(* Logix 5000 project; controller WWTP_SEC_CLX vendor 1 type 14 code 54 rev 17.2; software revision 17.00; part 9 of 13 *)
(* tags used below, declared in another part *)
   Inp_Faulted : BOOL;   // 1=Drive has Faulted (see drive display or manual)
   Inp_IntlkOK : BOOL;   // 1=Interlocks OK, drive can start/run
   Inp_NBIntlkOK : BOOL;   // 1=Non-Bypassable Interlocks OK, drive can start/run
   Inp_IOFault : BOOL;   // Input Communication Status 0=OK, 1=fail
   Inp_Sim : BOOL;   // 1=Simulate working drive; 0=Start/Stop/ Monitor actual drive
   Inp_Reset : BOOL;   // 1=Reset drive fault conditions and latched Alarms
   Cfg_HasOutDatalink : BOOL;   // 1=A signal is connected to Out_Datalink1
   Cfg_PCmdClear : BOOL;   // 1=Clear Program Commands on receipt 0=Leave Set
   Cfg_OvrdPermIntlk : BOOL;   // 1=Override ignores Bypassable Perm/ Intlk; 0=always use Perm/Intlk
   Cfg_HasFailToStartAlm : BOOL;   // 1=Fail to Start Alarm exists and will be checked
   Cfg_HasFailToStopAlm : BOOL;   // 1=Fail to Stop Alarm exists and will be checked
   Cfg_HasIntlkTripAlm : BOOL;   // 1=Interlock Trip Alarm exists and will be checked
   Cfg_HasDriveFaultAlm : BOOL;   // 1=Drive Fault alarm exists and will be checked
   Cfg_HasIOFaultAlm : BOOL;   // 1=I/O Fault Alarm exists and will be checked
   Cfg_FailToStartResetReqd : BOOL;   // 1=Reset requied to clear Fail to Start Alarm
   Cfg_FailToStopResetReqd : BOOL;   // 1=Reset required to clear Fail to Stop Alarm
   Cfg_IntlkTripResetReqd : BOOL;   // 1=Reset required to clear Interlock Trip Alarm
   Cfg_DriveFaultResetReqd : BOOL;   // 1=Reset required to clear Drive Fault Alarm
   Cfg_IOFaultResetReqd : BOOL;   // 1=Reset required to clear I/O Fault Alarm
   Cfg_FailToStartAckReqd : BOOL;   // 1=Acknowledge required for Fail to Start Alarm
   Cfg_FailToStopAckReqd : BOOL;   // 1=Acknowledge required for Fail to Stop Alarm
   Cfg_IntlkTripAckReqd : BOOL;   // 1=Acknowledge required for Interlock Trip Alarm
   Cfg_DriveFaultAckReqd : BOOL;   // 1=Acknowledge required for Drive Fault Alarm
   Cfg_IOFaultAckReqd : BOOL;   // 1=Acknowledge required for I/O Fault Alarm
   Cfg_FailToStartSeverity : SINT;   // Fail To Start Alarm Severity 1=info 2=warn 3=excep 4=fault
   Cfg_FailToStopSeverity : SINT;   // Fail To Stop Alarm Severity 1=info 2=warn 3=excep 4=fault
   Cfg_IntlkTripSeverity : SINT;   // Interlock Trip Alarm Severity 1=info 2=warn 3=excep 4=fault
   Cfg_DriveFaultSeverity : SINT;   // Drive Fault Alarm Severity 1=info, 2=warn, 3=excep, 4=fault
   Cfg_IOFaultSeverity : SINT;   // I/O Fault Alarm Severity 1=info 2=warn 3=excep 4=fault
   Cfg_MinSpdRef : REAL;   // Minimum Speed Reference in EU (for limiting)
   Cfg_MaxSpdRef : REAL;   // Maximum Speed Reference in EU (for limiting)
   Cfg_SpeedRefRawMin : INT;   // Speed Reference Minimum in Drive (raw) Units (for scaling)
   Cfg_SpeedRefRawMax : INT;   // Speed Reference Maximum in Drive (raw) Units (for scaling)
   Cfg_SpeedRefEUMin : REAL;   // Speed Reference Minimum in Engineering Units (for scaling)
   Cfg_SpeedRefEUMax : REAL;   // Speed Reference Maximum in Engineering Units (for scaling)
   Cfg_SpeedFdbkRawMin : INT;   // Speed Feedback Minimum in Drive (raw) Units (for scaling)
   Cfg_SpeedFdbkRawMax : INT;   // Speed Feedback Maximum in Drive (raw) Units (for scaling)
   Cfg_SpeedFdbkEUMin : REAL;   // Speed Feedback Minimum in Engineering Units (for scaling)
   Cfg_SpeedFdbkEUMax : REAL;   // Speed Feedback Maximum in Engineering Units (for scaling)
   Cfg_InpDatalinkRawMin : INT;   // Input Datalink Minimum in Drive (raw) Units (for scaling)
   Cfg_InpDatalinkRawMax : INT;   // Input Datalink Maximum in Drive (raw) Units (for scaling)
   Cfg_InpDatalinkEUMin : REAL;   // Input Datalink Minimum in Engineering Units (for scaling)
   Cfg_InpDatalinkEUMax : REAL;   // Input Datalink Maximum in Engineering Units (for scaling)
   Cfg_OutDatalinkMin : REAL;   // Minimum Output Datalink in EU (for limiting)
   Cfg_OutDatalinkMax : REAL;   // Maximum Output Datalink in EU (for limiting)
   Cfg_OutDatalinkRawMin : INT;   // Output Datalink Minimum in Drive (raw) Units (for scaling)
   Cfg_OutDatalinkRawMax : INT;   // Output Datalink Maximum in Drive (raw) Units (for scaling)
   Cfg_OutDatalinkEUMin : REAL;   // Output Datalink Minimum in Engineering Units (for scaling)
   Cfg_OutDatalinkEUMax : REAL;   // Output Datalink Maximum in Engineering Units (for scaling)
   PCmd_Reset : BOOL;   // Program Command to Reset drive fault and all Alarms requiring Reset
   PCmd_FailToStartAck : BOOL;   // Program Command to Acknowledge Fail to Start Alarm
   PCmd_FailToStartInhibit : BOOL;   // Program Command to Inhibit Fail to Start Alarm
   PCmd_FailToStartUninhibit : BOOL;   // Program Command to Uninhibit Fail to Start Alarm
   PCmd_FailToStopAck : BOOL;   // Program Command to Acknowledge Fail to Stop Alarm
   PCmd_FailToStopInhibit : BOOL;   // Program Command to Inhibit Fail to Stop Alarm
   PCmd_FailToStopUninhibit : BOOL;   // Program Command to Uninhibit Fail to Stop Alarm
   PCmd_IntlkTripAck : BOOL;   // Program Command to Acknowledge Interlock Trip Alarm
   PCmd_IntlkTripInhibit : BOOL;   // Program Command to Inhibit Interlock Trip Alarm
   PCmd_IntlkTripUninhibit : BOOL;   // Program Command to Uninhibit Interlock Trip Alarm
   PCmd_DriveFaultAck : BOOL;   // Program Command to Acknowledge Drive Fault Alarm
   PCmd_DriveFaultInhibit : BOOL;   // Program Command to Inhibit Drive Fault Alarm
   PCmd_DriveFaultUninhibit : BOOL;   // Program Command to Uninhibit Drive Fault Alarm
   PCmd_IOFaultAck : BOOL;   // Program Command to Acknowledge I/O Fault Alarm
   PCmd_IOFaultInhibit : BOOL;   // Program Command to Inhibit I/O Fault Alarm
   PCmd_IOFaultUninhibit : BOOL;   // Program Command to Uninhibit I/O Fault Alarm
   OCmd_Reset : BOOL;   // Operator Command to Reset all Alarms requiring Reset
   Out_SpeedRef : INT;   // Drive Speed Reference in Drive Units (typ. 0-32767 = 0 to max freq.)
   Out_Datalink : INT;   // Auxiliary Signal (datalink) Output in Drive (raw) Units
   Out_Run : BOOL;   // 1=Start/Run Drive, 0=Stop Drive (for held starter type)
   Out_Stop : BOOL;   // 1=Stop Drive, 0=drive left in current state
   Out_Start : BOOL;   // 1=Start Drive, 0=drive left in current state
   Out_Jog : BOOL;   // 1=Jog drive at Jog Speed, -->0=stop jogging
   Out_ClearFault : BOOL;   // 1=Attempt to clear Drive Fault
   Out_Fwd : BOOL;   // 1=Set drive direction to Forward
   Out_Rev : BOOL;   // 1=Set drive direction to Reverse
   Val_Notify : SINT;   // Current Alarm Level and Acknowledgement (enumeration)
   Sts_Disabled : BOOL;   // 1=Drive is Disabled
   Sts_Err : BOOL;   // 1=Error in Config: see detail bits for reason
   Err_Timer : BOOL;   // 1=Error in Config: Invalid Check or Reset Pulse Time (use 0 to 2147483)
   Err_Sim : BOOL;   // 1=Error in Config: simulation timer preset: use 0 to 2147483)
   Err_Alarm : BOOL;   // 1=Error in Config: Invalid Alarm Severity
   Err_FdbkRaw : BOOL;   // 1=Erron in Config: Speed Fdbk Raw Min = Max
   Err_FdbkEU : BOOL;   // 1=Error in Config: Speed Fdbk EU Min = Max
   Err_RefLim : BOOL;   // 1=Error in Config: Speed Ref Limit Min > Max
   Err_RefEU : BOOL;   // 1=Error in Config: Speed Ref EU Min = Max
   Err_RefRaw : BOOL;   // 1=Error in Config: Speed Ref Raw Min = Max
   Err_InpDLRaw : BOOL;   // 1=Error in Config: Input Datalink Raw Min = Max
   Err_InpDLEU : BOOL;   // 1=Error in Config: Input Datalink EU Min = Max
   Err_OutDLLim : BOOL;   // 1=Error in Config: Output Datalink Limits Min > Max
   Err_OutDLEU : BOOL;   // 1=Error in Config: Output Datalink EU Min = Max
   Err_OutDLRaw : BOOL;   // 1=Error in Config: Output Datalink Raw Min = Max
   Sts_Hand : BOOL;   // 1=Mode is Hand (supersedes Maint, Ovrd, Prog, Oper)
   Sts_Maint : BOOL;   // 1=Mode is Maintenance (supersedes Ovrd, Prog, Oper)
   Sts_Ovrd : BOOL;   // 1=Mode is Override (supersedes Prog, Oper)
   Sts_Prog : BOOL;   // 1=Mode is Program (auto)
   Sts_Oper : BOOL;   // 1=Mode is Operator (manual)
   Sts_ProgOperLock : BOOL;   // 1=Program or Operator has requested Mode Lock
   Sts_FailToStart : BOOL;   // 1=Drive Failed to Start (One-Shot)
   Alm_FailToStart : BOOL;   // 1=Drive Fail to tart Alarm
   Ack_FailToStart : BOOL;   // 1=Fail to Start Alarm has been acknowledged
   Sts_FailToStartDisabled : BOOL;   // 1=Fail to Start Alarm has been disabled (will not be sent)
   Sts_FailToStartInhibited : BOOL;   // 1=Fail to Start Alarm has been inhibited by logic
   Sts_FailToStartSuppressed : BOOL;   // 1=Fail to Start Alarm has been suppressed (logged only)
   Sts_FailToStop : BOOL;   // 1=Drive Failed to Stop
   Alm_FailToStop : BOOL;   // 1=Drive Fail to Stop Alarm
   Ack_FailToStop : BOOL;   // 1=Fail to Stop Alarm has been acknowledged
   Sts_FailToStopDisabled : BOOL;   // 1=Fail to Stop Alarm has been disabled (will not be sent)
   Sts_FailToStopInhibited : BOOL;   // 1=Fail to Stop Alarm has been inhibited by logic
   Sts_FailToStopSuppressed : BOOL;   // 1=Fail to Stop Alarm has been suppressed (logged only)
   Sts_IntlkTrip : BOOL;   // 1=Drive was stopped by an Interlock NOT OK (One-Shot)
   Alm_IntlkTrip : BOOL;   // 1=Alarm: Drive stopped by an Interlock NOT OK
   Ack_IntlkTrip : BOOL;   // 1=Interlock Trip Alarm has been acknowledged
   Sts_IntlkTripDisabled : BOOL;   // 1=Interlock Trip Alarm is Disabled (not saved or sent)
   Sts_IntlkTripInhibited : BOOL;   // 1=Interlock Trip Alarm has been inhibited by logic
   Sts_IntlkTripSuppressed : BOOL;   // 1=Interlock Trip Alarm has been suppressed (logged only)
   Sts_DriveFault : BOOL;   // 1=Drive Fault (see drive display or manual)
   Alm_DriveFault : BOOL;   // 1=Alarm: Drive Fault (see drive display or manual)
   Ack_DriveFault : BOOL;   // 1=Drive Fault Alarm has been acknowledged
   Sts_DriveFaultDisabled : BOOL;   // 1-=Drive Fault Alarm has been disabled (will not be sent)
   Sts_DriveFaultInhibited : BOOL;   // 1=Drive Fault Alarm has been inhibited by logic
   Sts_DriveFaultSuppressed : BOOL;   // 1-Drive Fault Alarm has been suppressed (logged only)
   Sts_IOFault : BOOL;   // I/O Comm Fault Status (0=OK, 1=Bad)
   Alm_IOFault : BOOL;   // 1=I/O Fault Alarm
   Ack_IOFault : BOOL;   // 1=I/O Fault Alarm has been acknowledged
   Sts_IOFaultDisabled : BOOL;   // 1=I/O Fault Alarm is Disabled (not saved or sent)
   Sts_IOFaultInhibited : BOOL;   // 1=I/O Fault Alarm has been inhibited by logic
   Sts_IOFaultSuppressed : BOOL;   // 1=I/O Fault Alarm has been suppressed (logged only)
   Rdy_Reset : BOOL;   // 1=Ready to receive OCmd_Reset (enables HMI button)
   Mode : P_Mode;   // Drive Mode Selection
   IOFault : P_Alarm;   // I/O Fault Alarm
   IntlkTrip : P_Alarm;   // Interlock Trip Alarm
   FailToStop : P_Alarm;   // Drive Failed to Stop Alarm
   FailToStart : P_Alarm;   // Drive Failed to Start Alarm
   Wrk_Run : BOOL;   // 1=Drive should be "running", 0=should be "stopped"
   Wrk_AccelT : TIMER;   // Simulation Accel Ramp timer until Running at speed
   Wrk_Fault : BOOL;   // 1=any Fault has been detected
   Wrk_DecelT : TIMER;   // Simulation Decel Ramp time until fully stopped
   Wrk_RunFdbk : BOOL;   // Run Feedback based on mode, simulation, etc. 1=running
   Wrk_IntlkTrip : BOOL;   // 1=Interlock Not OK Tripped Running Drive
   Wrk_Bypass : BOOL;   // Internal Bypassable Permissives and Interlocks are Bypassed flag
   Wrk_Disabled : BOOL;   // Internal Drive is Disabled
   DriveFault : P_Alarm;   // Drive Faulted Alarm
   Wrk_SpeedRef : REAL;   // Working copy of Speed Reference (for limiting)
   Wrk_Rev : BOOL;   // Working (internal) Direction 1=Reverse 0=Forward (default)
   Wrk_Jog : BOOL;   // 1=Jog Drive, 0=Drive not jogging
   Wrk_ResetT : TIMER;   // Reset Output Pulse Timer
   Wrk_ResetCond : BOOL;   // Any incoming Reset condition is TRUE
   Wrk_ResetONS : BOOL;   // One-Shot to fire Reset Timer to ensure min. output ON time.
   Wrk_OutDatalink : REAL;   // Selected Output Datalink setting
   Wrk_StopT : TIMER;   // Stop Check Timer (for Fail to Stop)
   Wrk_StartT : TIMER;   // Start Check Timer (for Fail to Start)
(* P_VSD, continued *)

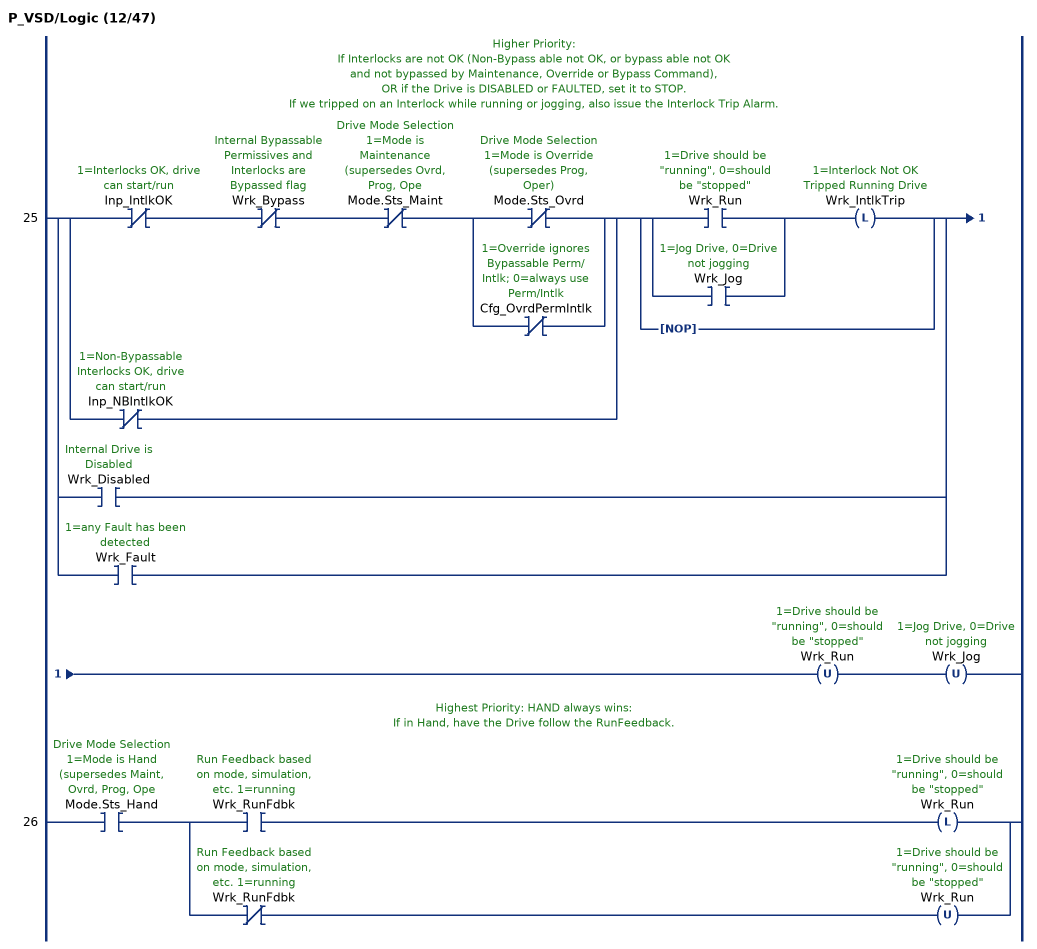
   [picture p171: P_VSD/Logic rungs 25-26]
   // Higher Priority:
   // If Interlocks are not OK (Non-Bypass able not OK, or bypass able not OK
   // and not bypassed by Maintenance, Override or Bypass Command),
   // OR if the Drive is DISABLED or FAULTED, set it to STOP.
   // If we tripped on an Interlock while running or jogging, also issue the Interlock Trip Alarm.
   25: [[XIO(Inp_IntlkOK) XIO(Wrk_Bypass) XIO(Mode.Sts_Maint) [XIO(Mode.Sts_Ovrd) ,XIO(Cfg_OvrdPermIntlk) ] ,XIO(Inp_NBIntlkOK) ] [[XIC(Wrk_Run) ,XIC(Wrk_Jog) ] OTL(Wrk_IntlkTrip) ,NOP() ] ,XIC(Wrk_Disabled) ,XIC(Wrk_Fault) ]OTU(Wrk_Run)OTU(Wrk_Jog);
   // Highest Priority: HAND always wins:
   // If in Hand, have the Drive follow the RunFeedback.
   26: XIC(Mode.Sts_Hand)[XIC(Wrk_RunFdbk) OTL(Wrk_Run) ,XIO(Wrk_RunFdbk) OTU(Wrk_Run) ];
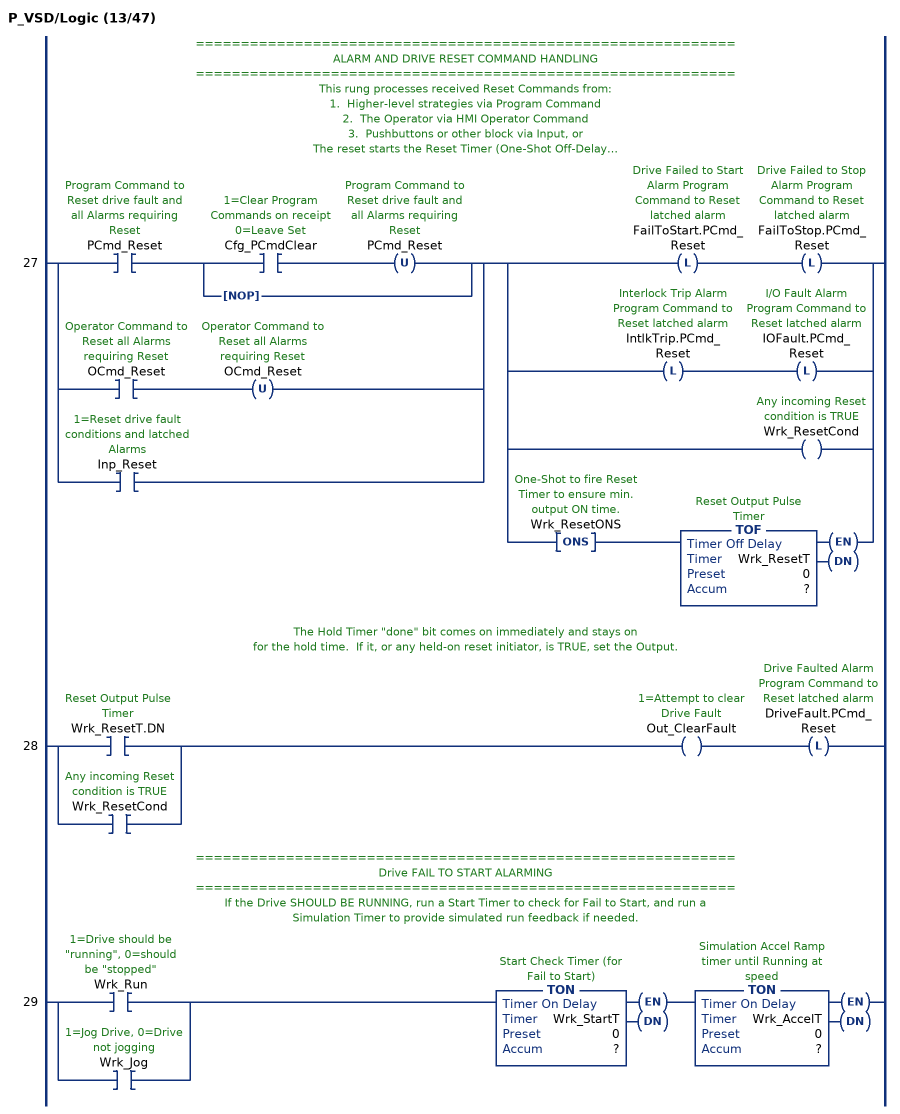
   // ============================================================
   // ALARM AND DRIVE RESET COMMAND HANDLING
   // ============================================================
   // This rung processes received Reset Commands from:
   // 1.  Higher-level strategies via Program Command
   // 2.  The Operator via HMI Operator Command
   // 3.  Pushbuttons or other block via Input, or
   // The reset starts the Reset Timer (One-Shot Off-Delay)
   // to ensure the output is held on for at least the minimum time.
   27: [XIC(PCmd_Reset) [XIC(Cfg_PCmdClear) OTU(PCmd_Reset) ,NOP() ] ,XIC(OCmd_Reset) OTU(OCmd_Reset) ,XIC(Inp_Reset) ][OTL(FailToStart.PCmd_Reset) OTL(FailToStop.PCmd_Reset) ,OTL(IntlkTrip.PCmd_Reset) OTL(IOFault.PCmd_Reset) ,OTE(Wrk_ResetCond) ,ONS(Wrk_ResetONS) TOF(Wrk_ResetT,?,?) ];
   // The Hold Timer "done" bit comes on immediately and stays on
   // for the hold time.  If it, or any held-on reset initiator, is TRUE, set the Output.
   28: [XIC(Wrk_ResetT.DN) ,XIC(Wrk_ResetCond) ]OTE(Out_ClearFault)OTL(DriveFault.PCmd_Reset);
   // ============================================================
   // Drive FAIL TO START ALARMING
   // ============================================================
   // If the Drive SHOULD BE RUNNING, run a Start Timer to check for Fail to Start, and run a
   // Simulation Timer to provide simulated run feedback if needed.
   29: [XIC(Wrk_Run) ,XIC(Wrk_Jog) ]TON(Wrk_StartT,?,?)TON(Wrk_AccelT,?,?);
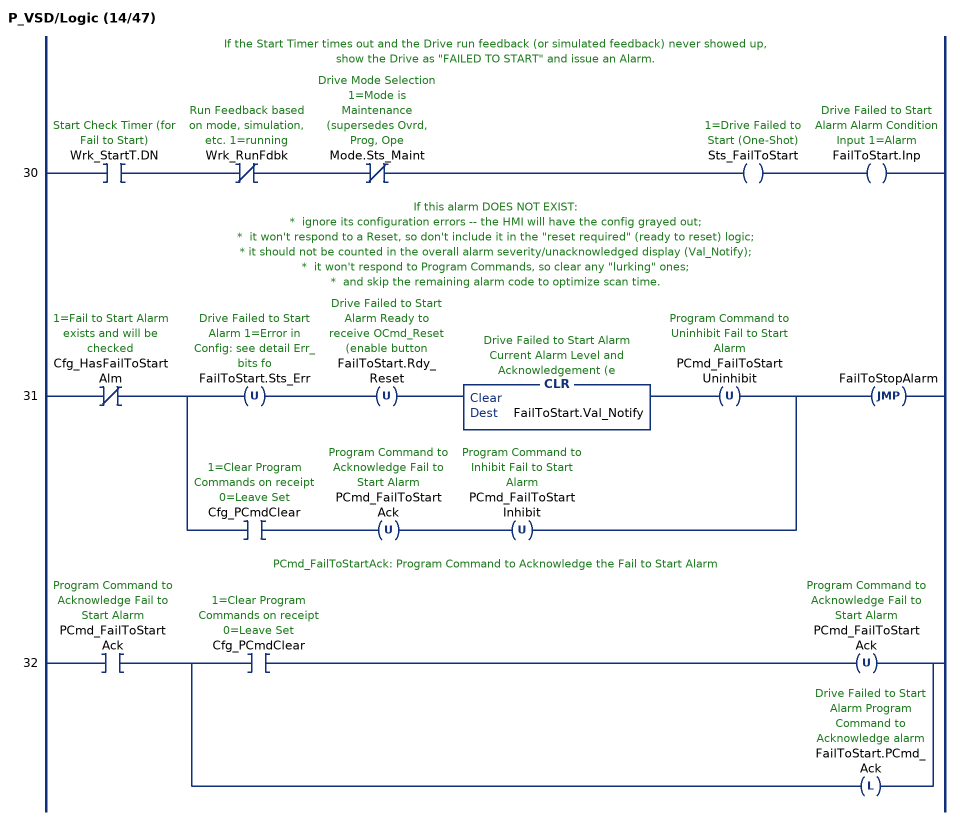
   // If the Start Timer times out and the Drive run feedback (or simulated feedback) never showed up,
   // show the Drive as "FAILED TO START" and issue an Alarm.
   30: XIC(Wrk_StartT.DN)XIO(Wrk_RunFdbk)XIO(Mode.Sts_Maint)OTE(Sts_FailToStart)OTE(FailToStart.Inp);
   // If this alarm DOES NOT EXIST:
   // *  ignore its configuration errors -- the HMI will have the config grayed out;
   // *  it won't respond to a Reset, so don't include it in the "reset required" (ready to reset) logic;
   // * it should not be counted in the overall alarm severity/unacknowledged display (Val_Notify);
   // *  it won't respond to Program Commands, so clear any "lurking" ones;
   // *  and skip the remaining alarm code to optimize scan time.
   31: XIO(Cfg_HasFailToStartAlm)[OTU(FailToStart.Sts_Err) OTU(FailToStart.Rdy_Reset) CLR(FailToStart.Val_Notify) OTU(PCmd_FailToStartUninhibit) ,XIC(Cfg_PCmdClear) OTU(PCmd_FailToStartAck) OTU(PCmd_FailToStartInhibit) ]JMP(FailToStopAlarm);
   // PCmd_FailToStartAck: Program Command to Acknowledge the Fail to Start Alarm
   32: XIC(PCmd_FailToStartAck)[XIC(Cfg_PCmdClear) OTU(PCmd_FailToStartAck) ,OTL(FailToStart.PCmd_Ack) ];
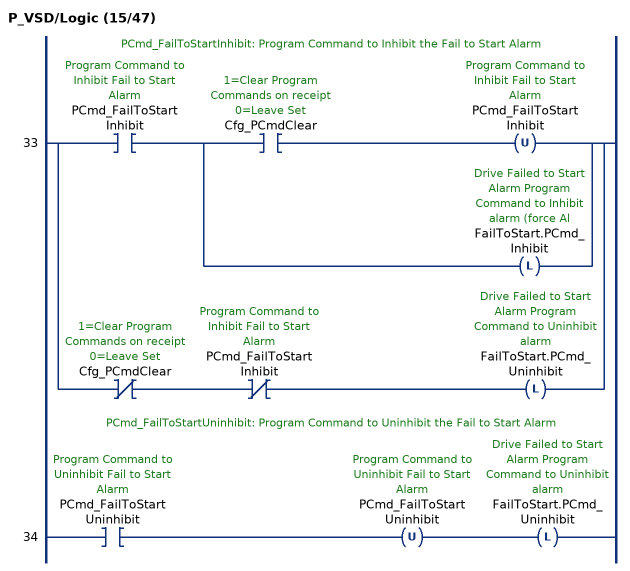
   // PCmd_FailToStartInhibit: Program Command to Inhibit the Fail to Start Alarm
   33: [XIC(PCmd_FailToStartInhibit) [XIC(Cfg_PCmdClear) OTU(PCmd_FailToStartInhibit) ,OTL(FailToStart.PCmd_Inhibit) ] ,XIO(Cfg_PCmdClear) XIO(PCmd_FailToStartInhibit) OTL(FailToStart.PCmd_Uninhibit) ];
   // PCmd_FailToStartUninhibit: Program Command to Uninhibit the Fail to Start Alarm
   34: XIC(PCmd_FailToStartUninhibit)OTU(PCmd_FailToStartUninhibit)OTL(FailToStart.PCmd_Uninhibit);
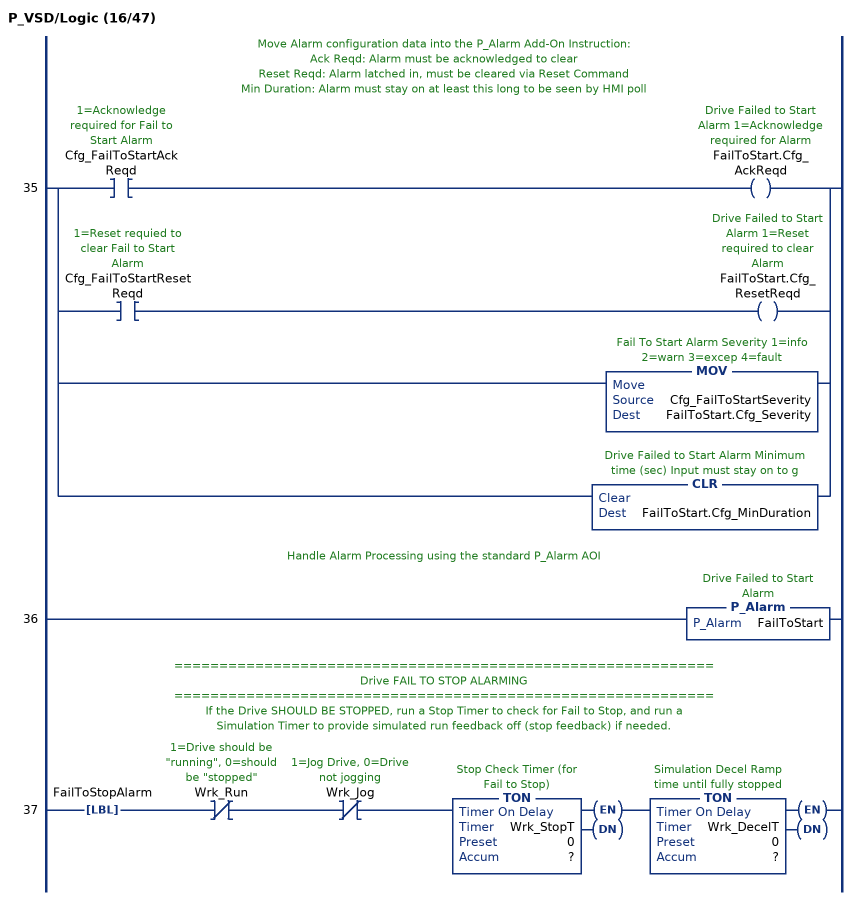
   // Move Alarm configuration data into the P_Alarm Add-On Instruction:
   // Ack Reqd: Alarm must be acknowledged to clear
   // Reset Reqd: Alarm latched in, must be cleared via Reset Command
   // Min Duration: Alarm must stay on at least this long to be seen by HMI poll
   35: [XIC(Cfg_FailToStartAckReqd) OTE(FailToStart.Cfg_AckReqd) ,XIC(Cfg_FailToStartResetReqd) OTE(FailToStart.Cfg_ResetReqd) ,MOV(Cfg_FailToStartSeverity,FailToStart.Cfg_Severity) ,CLR(FailToStart.Cfg_MinDuration) ];
   // Handle Alarm Processing using the standard P_Alarm AOI
   36: P_Alarm(FailToStart);
   // ============================================================
   // Drive FAIL TO STOP ALARMING
   // ============================================================
   // If the Drive SHOULD BE STOPPED, run a Stop Timer to check for Fail to Stop, and run a
   // Simulation Timer to provide simulated run feedback off (stop feedback) if needed.
   37: LBL(FailToStopAlarm)XIO(Wrk_Run)XIO(Wrk_Jog)TON(Wrk_StopT,?,?)TON(Wrk_DecelT,?,?);
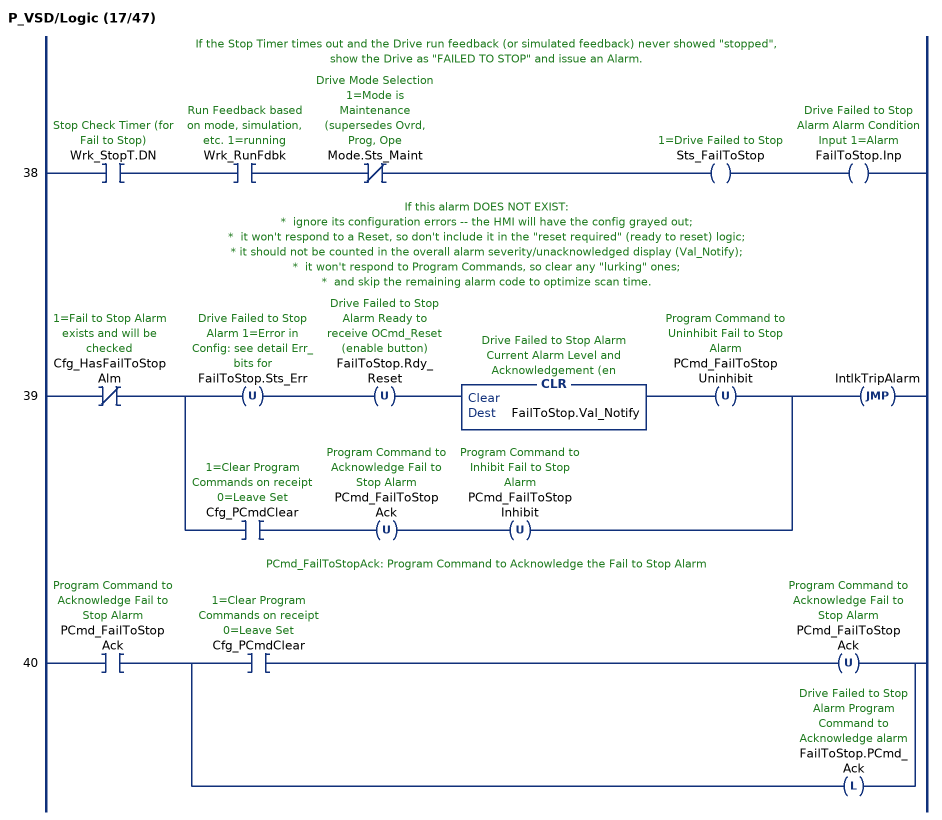
   // If the Stop Timer times out and the Drive run feedback (or simulated feedback) never showed "stopped",
   // show the Drive as "FAILED TO STOP" and issue an Alarm.
   38: XIC(Wrk_StopT.DN)XIC(Wrk_RunFdbk)XIO(Mode.Sts_Maint)OTE(Sts_FailToStop)OTE(FailToStop.Inp);
   // If this alarm DOES NOT EXIST:
   // *  ignore its configuration errors -- the HMI will have the config grayed out;
   // *  it won't respond to a Reset, so don't include it in the "reset required" (ready to reset) logic;
   // * it should not be counted in the overall alarm severity/unacknowledged display (Val_Notify);
   // *  it won't respond to Program Commands, so clear any "lurking" ones;
   // *  and skip the remaining alarm code to optimize scan time.
   39: XIO(Cfg_HasFailToStopAlm)[OTU(FailToStop.Sts_Err) OTU(FailToStop.Rdy_Reset) CLR(FailToStop.Val_Notify) OTU(PCmd_FailToStopUninhibit) ,XIC(Cfg_PCmdClear) OTU(PCmd_FailToStopAck) OTU(PCmd_FailToStopInhibit) ]JMP(IntlkTripAlarm);
   // PCmd_FailToStopAck: Program Command to Acknowledge the Fail to Stop Alarm
   40: XIC(PCmd_FailToStopAck)[XIC(Cfg_PCmdClear) OTU(PCmd_FailToStopAck) ,OTL(FailToStop.PCmd_Ack) ];
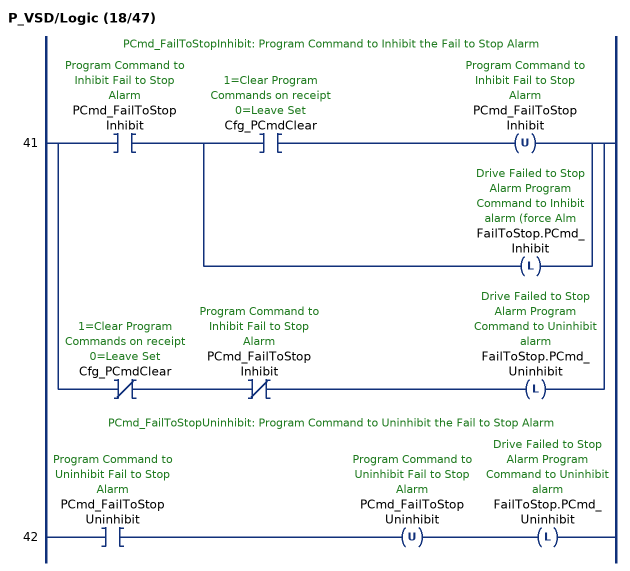
   // PCmd_FailToStopInhibit: Program Command to Inhibit the Fail to Stop Alarm
   41: [XIC(PCmd_FailToStopInhibit) [XIC(Cfg_PCmdClear) OTU(PCmd_FailToStopInhibit) ,OTL(FailToStop.PCmd_Inhibit) ] ,XIO(Cfg_PCmdClear) XIO(PCmd_FailToStopInhibit) OTL(FailToStop.PCmd_Uninhibit) ];
   // PCmd_FailToStopUninhibit: Program Command to Uninhibit the Fail to Stop Alarm
   42: XIC(PCmd_FailToStopUninhibit)OTU(PCmd_FailToStopUninhibit)OTL(FailToStop.PCmd_Uninhibit);
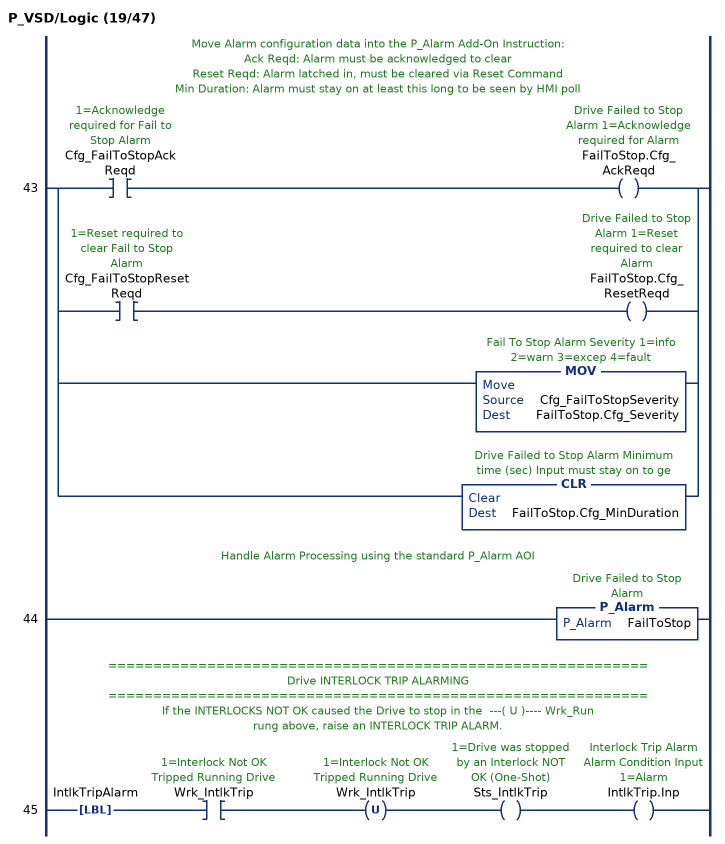
   // Move Alarm configuration data into the P_Alarm Add-On Instruction:
   // Ack Reqd: Alarm must be acknowledged to clear
   // Reset Reqd: Alarm latched in, must be cleared via Reset Command
   // Min Duration: Alarm must stay on at least this long to be seen by HMI poll
   43: [XIC(Cfg_FailToStopAckReqd) OTE(FailToStop.Cfg_AckReqd) ,XIC(Cfg_FailToStopResetReqd) OTE(FailToStop.Cfg_ResetReqd) ,MOV(Cfg_FailToStopSeverity,FailToStop.Cfg_Severity) ,CLR(FailToStop.Cfg_MinDuration) ];
   // Handle Alarm Processing using the standard P_Alarm AOI
   44: P_Alarm(FailToStop);
   // ============================================================
   // Drive INTERLOCK TRIP ALARMING
   // ============================================================
   // If the INTERLOCKS NOT OK caused the Drive to stop in the  ---( U )---- Wrk_Run
   // rung above, raise an INTERLOCK TRIP ALARM.
   45: LBL(IntlkTripAlarm)XIC(Wrk_IntlkTrip)OTU(Wrk_IntlkTrip)OTE(Sts_IntlkTrip)OTE(IntlkTrip.Inp);
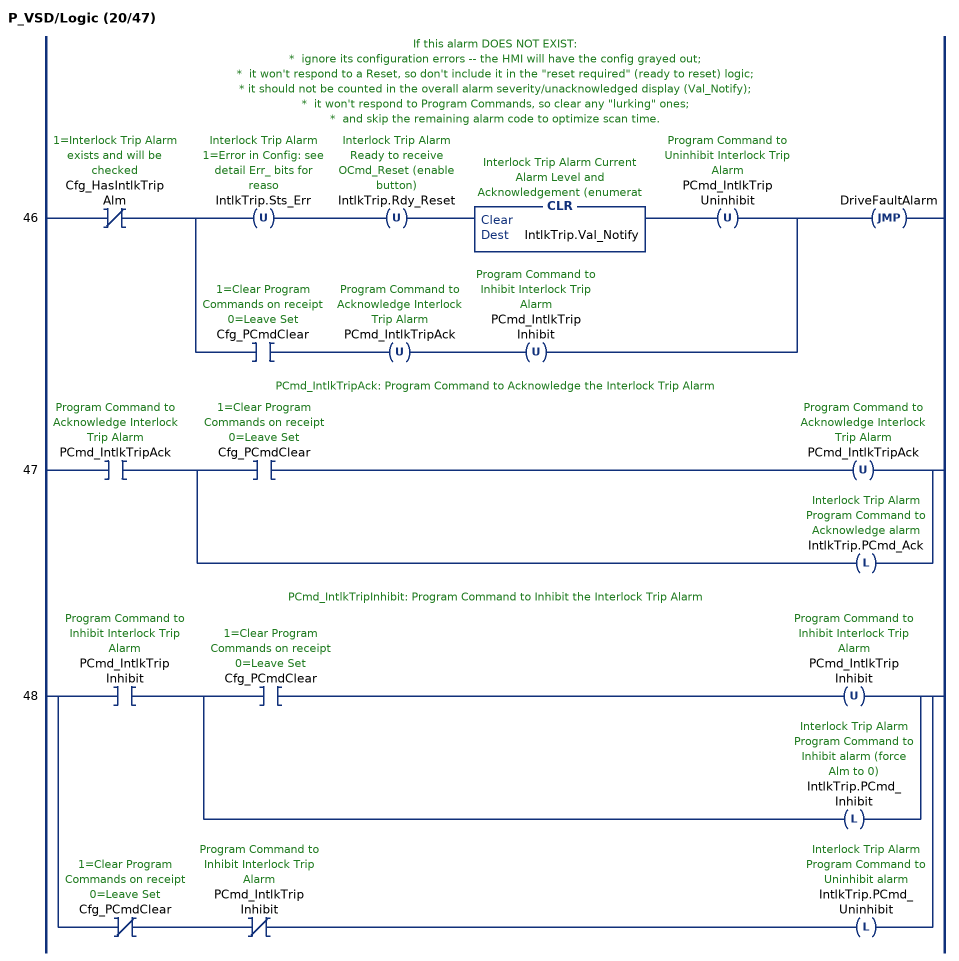
   // If this alarm DOES NOT EXIST:
   // *  ignore its configuration errors -- the HMI will have the config grayed out;
   // *  it won't respond to a Reset, so don't include it in the "reset required" (ready to reset) logic;
   // * it should not be counted in the overall alarm severity/unacknowledged display (Val_Notify);
   // *  it won't respond to Program Commands, so clear any "lurking" ones;
   // *  and skip the remaining alarm code to optimize scan time.
   46: XIO(Cfg_HasIntlkTripAlm)[OTU(IntlkTrip.Sts_Err) OTU(IntlkTrip.Rdy_Reset) CLR(IntlkTrip.Val_Notify) OTU(PCmd_IntlkTripUninhibit) ,XIC(Cfg_PCmdClear) OTU(PCmd_IntlkTripAck) OTU(PCmd_IntlkTripInhibit) ]JMP(DriveFaultAlarm);
   // PCmd_IntlkTripAck: Program Command to Acknowledge the Interlock Trip Alarm
   47: XIC(PCmd_IntlkTripAck)[XIC(Cfg_PCmdClear) OTU(PCmd_IntlkTripAck) ,OTL(IntlkTrip.PCmd_Ack) ];
   // PCmd_IntlkTripInhibit: Program Command to Inhibit the Interlock Trip Alarm
   48: [XIC(PCmd_IntlkTripInhibit) [XIC(Cfg_PCmdClear) OTU(PCmd_IntlkTripInhibit) ,OTL(IntlkTrip.PCmd_Inhibit) ] ,XIO(Cfg_PCmdClear) XIO(PCmd_IntlkTripInhibit) OTL(IntlkTrip.PCmd_Uninhibit) ];
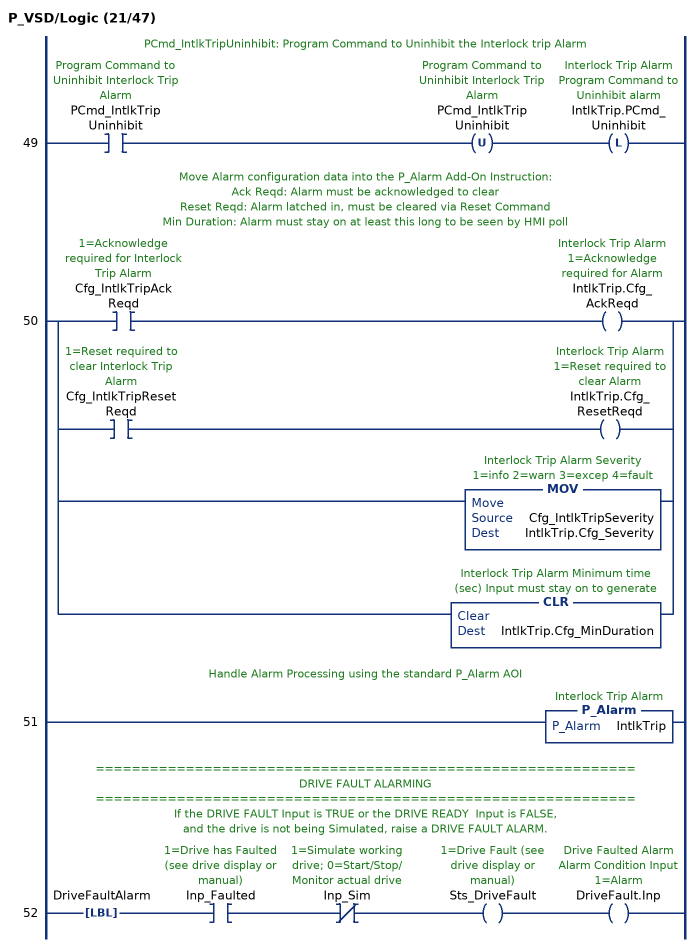
   // PCmd_IntlkTripUninhibit: Program Command to Uninhibit the Interlock trip Alarm
   49: XIC(PCmd_IntlkTripUninhibit)OTU(PCmd_IntlkTripUninhibit)OTL(IntlkTrip.PCmd_Uninhibit);
   // Move Alarm configuration data into the P_Alarm Add-On Instruction:
   // Ack Reqd: Alarm must be acknowledged to clear
   // Reset Reqd: Alarm latched in, must be cleared via Reset Command
   // Min Duration: Alarm must stay on at least this long to be seen by HMI poll
   50: [XIC(Cfg_IntlkTripAckReqd) OTE(IntlkTrip.Cfg_AckReqd) ,XIC(Cfg_IntlkTripResetReqd) OTE(IntlkTrip.Cfg_ResetReqd) ,MOV(Cfg_IntlkTripSeverity,IntlkTrip.Cfg_Severity) ,CLR(IntlkTrip.Cfg_MinDuration) ];
   // Handle Alarm Processing using the standard P_Alarm AOI
   51: P_Alarm(IntlkTrip);
   // ============================================================
   // DRIVE FAULT ALARMING
   // ============================================================
   // If the DRIVE FAULT Input is TRUE or the DRIVE READY  Input is FALSE,
   // and the drive is not being Simulated, raise a DRIVE FAULT ALARM.
   52: LBL(DriveFaultAlarm)XIC(Inp_Faulted)XIO(Inp_Sim)OTE(Sts_DriveFault)OTE(DriveFault.Inp);
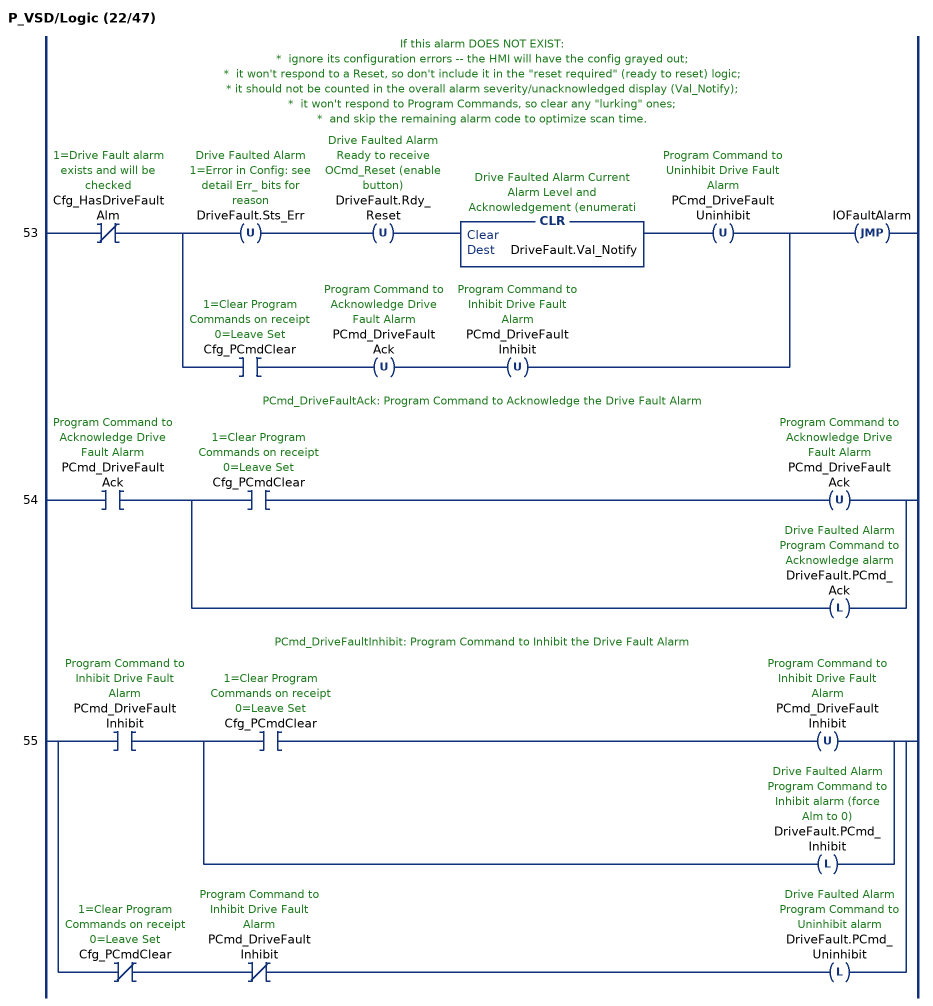
   // If this alarm DOES NOT EXIST:
   // *  ignore its configuration errors -- the HMI will have the config grayed out;
   // *  it won't respond to a Reset, so don't include it in the "reset required" (ready to reset) logic;
   // * it should not be counted in the overall alarm severity/unacknowledged display (Val_Notify);
   // *  it won't respond to Program Commands, so clear any "lurking" ones;
   // *  and skip the remaining alarm code to optimize scan time.
   53: XIO(Cfg_HasDriveFaultAlm)[OTU(DriveFault.Sts_Err) OTU(DriveFault.Rdy_Reset) CLR(DriveFault.Val_Notify) OTU(PCmd_DriveFaultUninhibit) ,XIC(Cfg_PCmdClear) OTU(PCmd_DriveFaultAck) OTU(PCmd_DriveFaultInhibit) ]JMP(IOFaultAlarm);
   // PCmd_DriveFaultAck: Program Command to Acknowledge the Drive Fault Alarm
   54: XIC(PCmd_DriveFaultAck)[XIC(Cfg_PCmdClear) OTU(PCmd_DriveFaultAck) ,OTL(DriveFault.PCmd_Ack) ];
   // PCmd_DriveFaultInhibit: Program Command to Inhibit the Drive Fault Alarm
   55: [XIC(PCmd_DriveFaultInhibit) [XIC(Cfg_PCmdClear) OTU(PCmd_DriveFaultInhibit) ,OTL(DriveFault.PCmd_Inhibit) ] ,XIO(Cfg_PCmdClear) XIO(PCmd_DriveFaultInhibit) OTL(DriveFault.PCmd_Uninhibit) ];
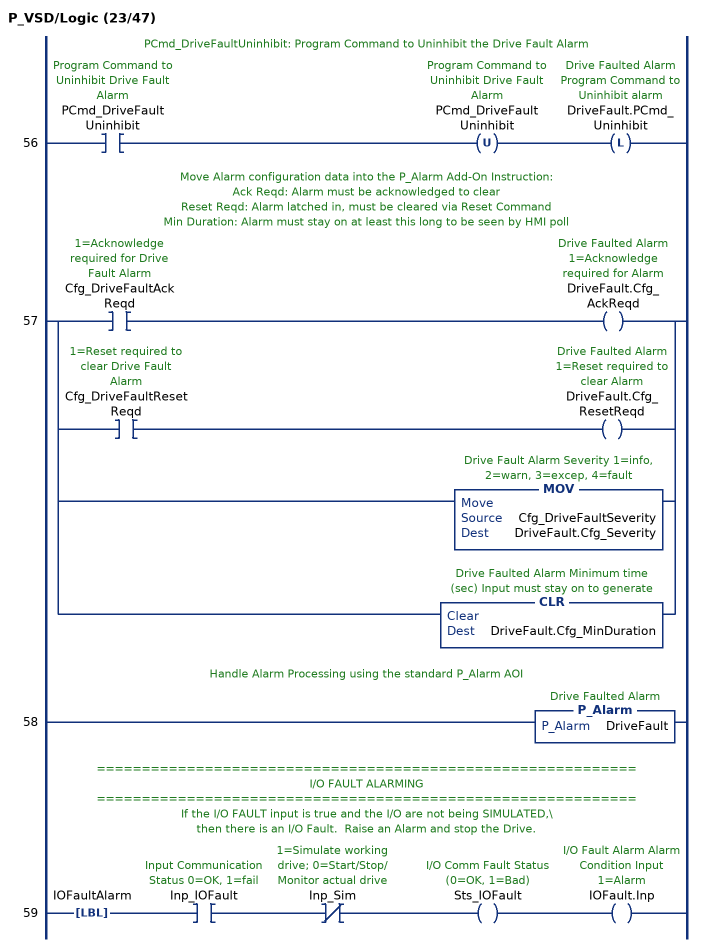
   // PCmd_DriveFaultUninhibit: Program Command to Uninhibit the Drive Fault Alarm
   56: XIC(PCmd_DriveFaultUninhibit)OTU(PCmd_DriveFaultUninhibit)OTL(DriveFault.PCmd_Uninhibit);
   // Move Alarm configuration data into the P_Alarm Add-On Instruction:
   // Ack Reqd: Alarm must be acknowledged to clear
   // Reset Reqd: Alarm latched in, must be cleared via Reset Command
   // Min Duration: Alarm must stay on at least this long to be seen by HMI poll
   57: [XIC(Cfg_DriveFaultAckReqd) OTE(DriveFault.Cfg_AckReqd) ,XIC(Cfg_DriveFaultResetReqd) OTE(DriveFault.Cfg_ResetReqd) ,MOV(Cfg_DriveFaultSeverity,DriveFault.Cfg_Severity) ,CLR(DriveFault.Cfg_MinDuration) ];
   // Handle Alarm Processing using the standard P_Alarm AOI
   58: P_Alarm(DriveFault);
   // ============================================================
   // I/O FAULT ALARMING
   // ============================================================
   // If the I/O FAULT input is true and the I/O are not being SIMULATED,\
   // then there is an I/O Fault.  Raise an Alarm and stop the Drive.
   59: LBL(IOFaultAlarm)XIC(Inp_IOFault)XIO(Inp_Sim)OTE(Sts_IOFault)OTE(IOFault.Inp);
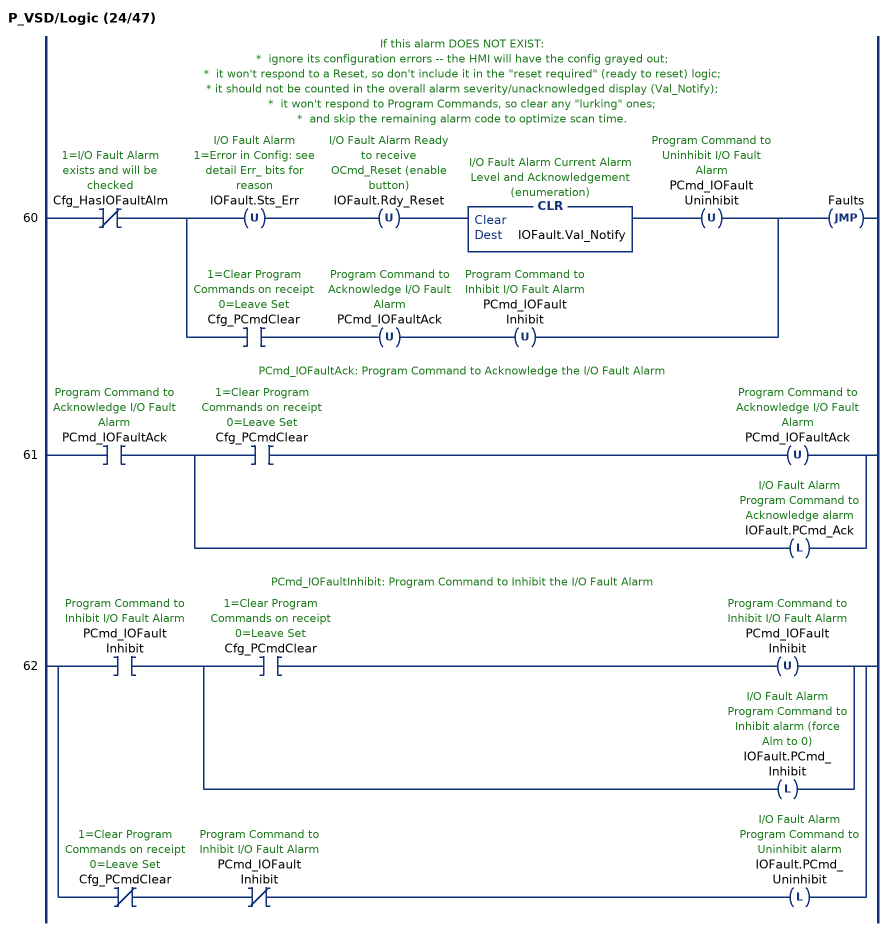
   // If this alarm DOES NOT EXIST:
   // *  ignore its configuration errors -- the HMI will have the config grayed out;
   // *  it won't respond to a Reset, so don't include it in the "reset required" (ready to reset) logic;
   // * it should not be counted in the overall alarm severity/unacknowledged display (Val_Notify);
   // *  it won't respond to Program Commands, so clear any "lurking" ones;
   // *  and skip the remaining alarm code to optimize scan time.
   60: XIO(Cfg_HasIOFaultAlm)[OTU(IOFault.Sts_Err) OTU(IOFault.Rdy_Reset) CLR(IOFault.Val_Notify) OTU(PCmd_IOFaultUninhibit) ,XIC(Cfg_PCmdClear) OTU(PCmd_IOFaultAck) OTU(PCmd_IOFaultInhibit) ]JMP(Faults);
   // PCmd_IOFaultAck: Program Command to Acknowledge the I/O Fault Alarm
   61: XIC(PCmd_IOFaultAck)[XIC(Cfg_PCmdClear) OTU(PCmd_IOFaultAck) ,OTL(IOFault.PCmd_Ack) ];
   // PCmd_IOFaultInhibit: Program Command to Inhibit the I/O Fault Alarm
   62: [XIC(PCmd_IOFaultInhibit) [XIC(Cfg_PCmdClear) OTU(PCmd_IOFaultInhibit) ,OTL(IOFault.PCmd_Inhibit) ] ,XIO(Cfg_PCmdClear) XIO(PCmd_IOFaultInhibit) OTL(IOFault.PCmd_Uninhibit) ];
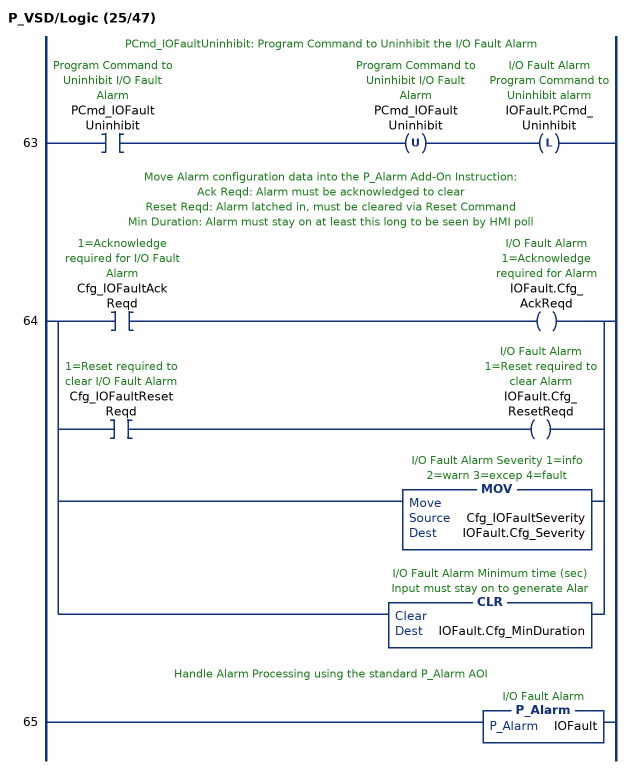
   // PCmd_IOFaultUninhibit: Program Command to Uninhibit the I/O Fault Alarm
   63: XIC(PCmd_IOFaultUninhibit)OTU(PCmd_IOFaultUninhibit)OTL(IOFault.PCmd_Uninhibit);
   // Move Alarm configuration data into the P_Alarm Add-On Instruction:
   // Ack Reqd: Alarm must be acknowledged to clear
   // Reset Reqd: Alarm latched in, must be cleared via Reset Command
   // Min Duration: Alarm must stay on at least this long to be seen by HMI poll
   64: [XIC(Cfg_IOFaultAckReqd) OTE(IOFault.Cfg_AckReqd) ,XIC(Cfg_IOFaultResetReqd) OTE(IOFault.Cfg_ResetReqd) ,MOV(Cfg_IOFaultSeverity,IOFault.Cfg_Severity) ,CLR(IOFault.Cfg_MinDuration) ];
   // Handle Alarm Processing using the standard P_Alarm AOI
   65: P_Alarm(IOFault);
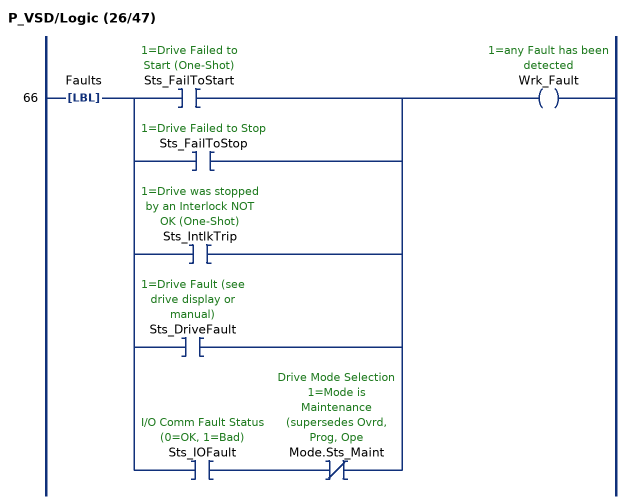
   66: LBL(Faults)[XIC(Sts_FailToStart) ,XIC(Sts_FailToStop) ,XIC(Sts_IntlkTrip) ,XIC(Sts_DriveFault) ,XIC(Sts_IOFault) XIO(Mode.Sts_Maint) ]OTE(Wrk_Fault);
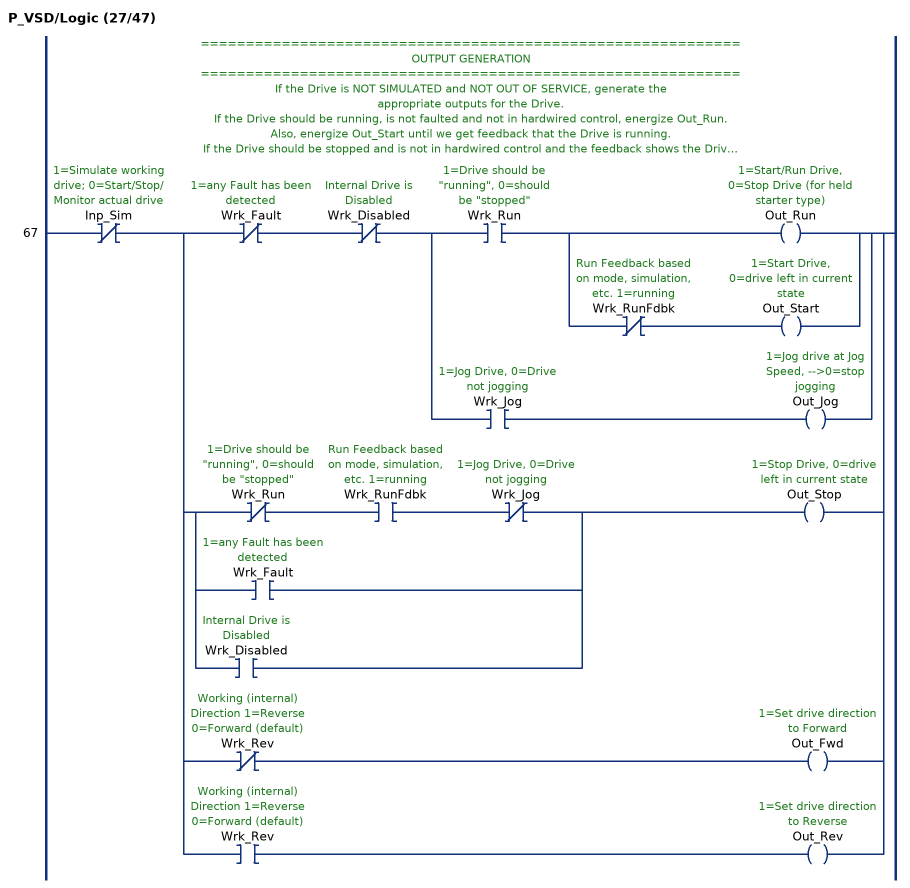
   // ============================================================
   // OUTPUT GENERATION
   // ============================================================
   // If the Drive is NOT SIMULATED and NOT OUT OF SERVICE, generate the
   // appropriate outputs for the Drive.
   // If the Drive should be running, is not faulted and not in hardwired control, energize Out_Run.
   // Also, energize Out_Start until we get feedback that the Drive is running.
   // If the Drive should be stopped and is not in hardwired control and the feedback shows the Drive
   // is NOT stopped, or if the Drive is Faulted, energize the Out_Stop output to stop the Drive.
   67: XIO(Inp_Sim)[XIO(Wrk_Fault) XIO(Wrk_Disabled) [XIC(Wrk_Run) [OTE(Out_Run) ,XIO(Wrk_RunFdbk) OTE(Out_Start) ] ,XIC(Wrk_Jog) OTE(Out_Jog) ] ,[XIO(Wrk_Run) XIC(Wrk_RunFdbk) XIO(Wrk_Jog) ,XIC(Wrk_Fault) ,XIC(Wrk_Disabled) ] OTE(Out_Stop) ,XIO(Wrk_Rev) OTE(Out_Fwd) ,XIC(Wrk_Rev) OTE(Out_Rev) ];
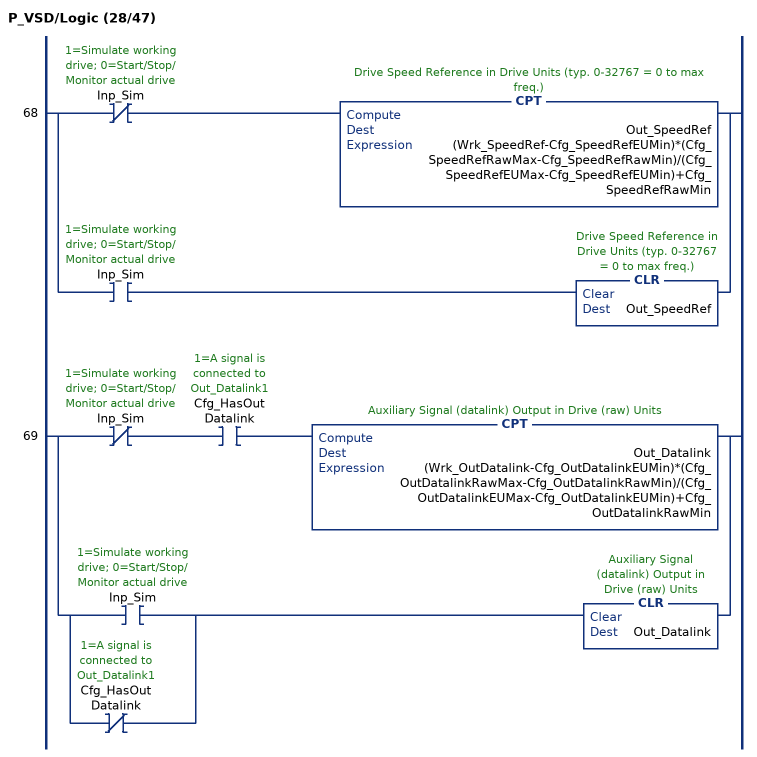
   68: [XIO(Inp_Sim) CPT(Out_SpeedRef,(Wrk_SpeedRef-Cfg_SpeedRefEUMin)*(Cfg_SpeedRefRawMax-Cfg_SpeedRefRawMin)/(Cfg_SpeedRefEUMax-Cfg_SpeedRefEUMin)+Cfg_SpeedRefRawMin) ,XIC(Inp_Sim) CLR(Out_SpeedRef) ];
   69: [XIO(Inp_Sim) XIC(Cfg_HasOutDatalink) CPT(Out_Datalink,(Wrk_OutDatalink-Cfg_OutDatalinkEUMin)*(Cfg_OutDatalinkRawMax-Cfg_OutDatalinkRawMin)/(Cfg_OutDatalinkEUMax-Cfg_OutDatalinkEUMin)+Cfg_OutDatalinkRawMin) ,[XIC(Inp_Sim) ,XIO(Cfg_HasOutDatalink) ] CLR(Out_Datalink) ];
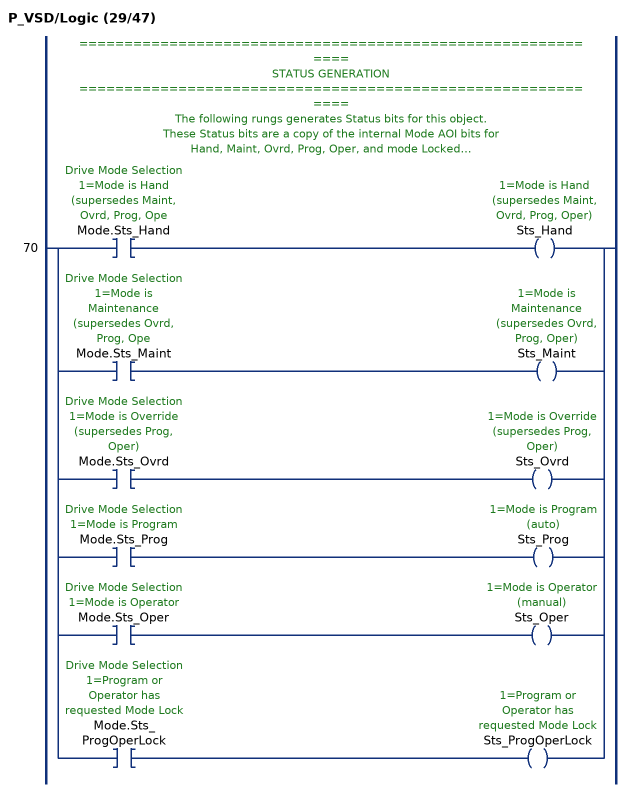
   // ============================================================
   // STATUS GENERATION
   // ============================================================
   // The following rungs generates Status bits for this object.
   // These Status bits are a copy of the internal Mode AOI bits for
   // Hand, Maint, Ovrd, Prog, Oper, and mode Locked.
   // NOTE for Sts_Maint:  This Drive is in Maintenance (Out Of Service, no able to run normally)
   // if this instruction is on a False Rung (Enable In False).  See the Enable In False Routine.
   70: [XIC(Mode.Sts_Hand) OTE(Sts_Hand) ,XIC(Mode.Sts_Maint) OTE(Sts_Maint) ,XIC(Mode.Sts_Ovrd) OTE(Sts_Ovrd) ,XIC(Mode.Sts_Prog) OTE(Sts_Prog) ,XIC(Mode.Sts_Oper) OTE(Sts_Oper) ,XIC(Mode.Sts_ProgOperLock) OTE(Sts_ProgOperLock) ];
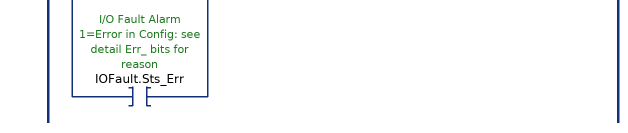
   // This rung handles the reports of all Bad Configuration Status.
   // Individual bits are provided for various status:
   // Bad Raw Scaling configs
   // Bad Engineering Units Scaling configs
   // Bad 1st-Order Filter configs
   // Bad Alarm Dead band configs
   // Bad Alarm Minimum Duration configs
   // Then a summary Bad Config status is provided, simply an OR of the individual bits.
   71: [EQU(Cfg_SpeedFdbkRawMax,Cfg_SpeedFdbkRawMin) OTE(Err_FdbkRaw) ,EQU(Cfg_SpeedFdbkEUMax,Cfg_SpeedFdbkEUMin) OTE(Err_FdbkEU) ,EQU(Cfg_MaxSpdRef,Cfg_MinSpdRef) OTE(Err_RefLim) ,EQU(Cfg_SpeedRefEUMax,Cfg_SpeedRefEUMin) OTE(Err_RefEU) ,EQU(Cfg_SpeedRefRawMax,Cfg_SpeedRefRawMin) OTE(Err_RefRaw) ,EQU(Cfg_InpDatalinkRawMax,Cfg_InpDatalinkRawMin) OTE(Err_InpDLRaw) ,EQU(Cfg_InpDatalinkEUMax,Cfg_InpDatalinkEUMin) OTE(Err_InpDLEU) ,EQU(Cfg_OutDatalinkMax,Cfg_OutDatalinkMin) OTE(Err_OutDLLim) ,EQU(Cfg_OutDatalinkEUMax,Cfg_OutDatalinkEUMin) OTE(Err_OutDLEU) ,EQU(Cfg_OutDatalinkRawMax,Cfg_OutDatalinkRawMin) OTE(Err_OutDLRaw) ,XIC(Err_Timer) ,XIC(Err_Sim) ,[XIC(FailToStart.Sts_Err) ,XIC(FailToStop.Sts_Err) ,XIC(IntlkTrip.Sts_Err) ,XIC(DriveFault.Sts_Err) ,XIC(IOFault.Sts_Err) ] OTE(Err_Alarm) ]OTE(Sts_Err);
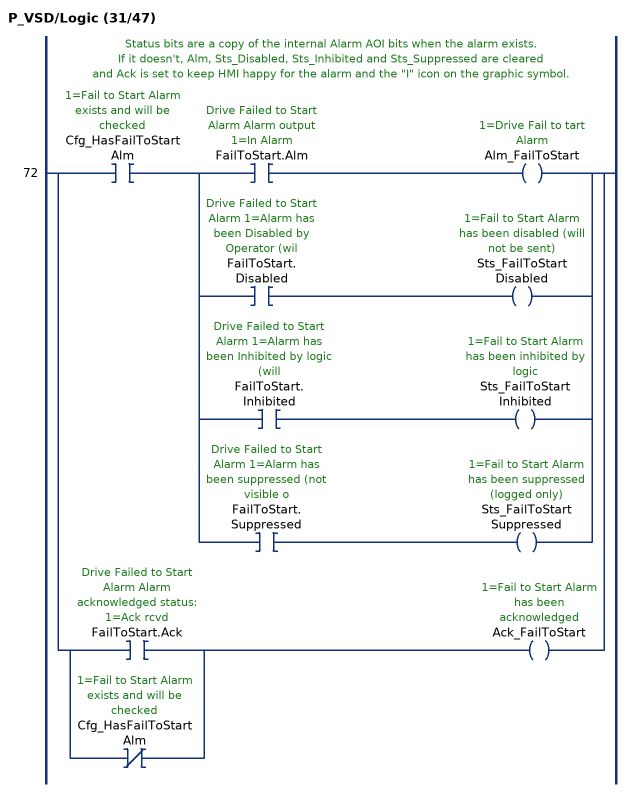
   // Status bits are a copy of the internal Alarm AOI bits when the alarm exists.
   // If it doesn't, Alm, Sts_Disabled, Sts_Inhibited and Sts_Suppressed are cleared
   // and Ack is set to keep HMI happy for the alarm and the "I" icon on the graphic symbol.
   72: [XIC(Cfg_HasFailToStartAlm) [XIC(FailToStart.Alm) OTE(Alm_FailToStart) ,XIC(FailToStart.Disabled) OTE(Sts_FailToStartDisabled) ,XIC(FailToStart.Inhibited) OTE(Sts_FailToStartInhibited) ,XIC(FailToStart.Suppressed) OTE(Sts_FailToStartSuppressed) ] ,[XIC(FailToStart.Ack) ,XIO(Cfg_HasFailToStartAlm) ] OTE(Ack_FailToStart) ];
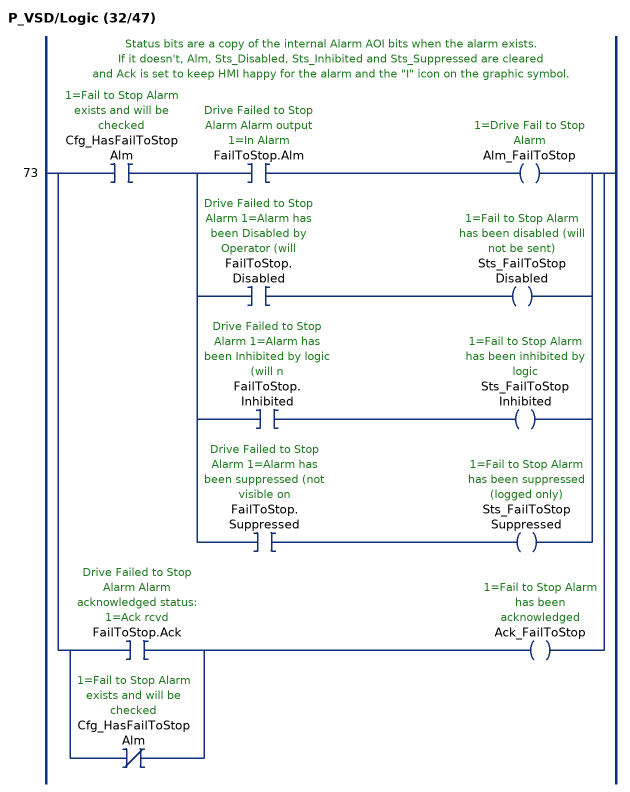
   // Status bits are a copy of the internal Alarm AOI bits when the alarm exists.
   // If it doesn't, Alm, Sts_Disabled, Sts_Inhibited and Sts_Suppressed are cleared
   // and Ack is set to keep HMI happy for the alarm and the "I" icon on the graphic symbol.
   73: [XIC(Cfg_HasFailToStopAlm) [XIC(FailToStop.Alm) OTE(Alm_FailToStop) ,XIC(FailToStop.Disabled) OTE(Sts_FailToStopDisabled) ,XIC(FailToStop.Inhibited) OTE(Sts_FailToStopInhibited) ,XIC(FailToStop.Suppressed) OTE(Sts_FailToStopSuppressed) ] ,[XIC(FailToStop.Ack) ,XIO(Cfg_HasFailToStopAlm) ] OTE(Ack_FailToStop) ];
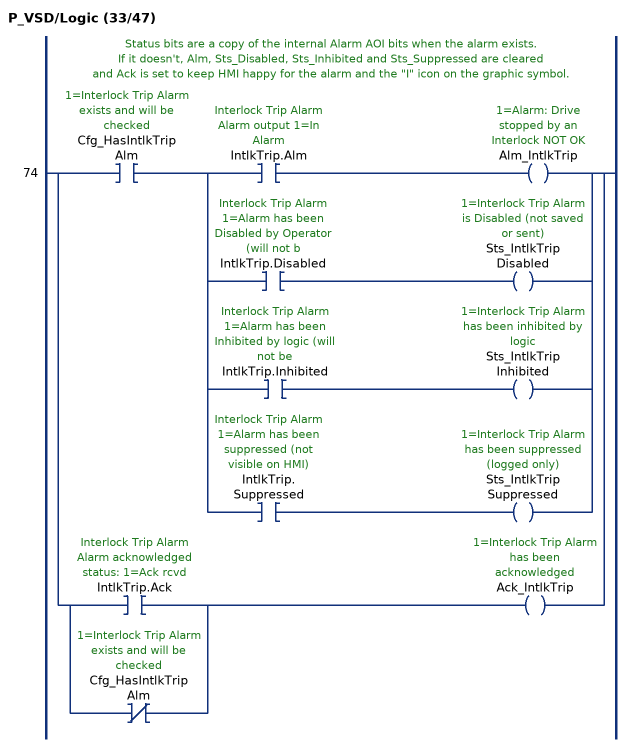
   // Status bits are a copy of the internal Alarm AOI bits when the alarm exists.
   // If it doesn't, Alm, Sts_Disabled, Sts_Inhibited and Sts_Suppressed are cleared
   // and Ack is set to keep HMI happy for the alarm and the "I" icon on the graphic symbol.
   74: [XIC(Cfg_HasIntlkTripAlm) [XIC(IntlkTrip.Alm) OTE(Alm_IntlkTrip) ,XIC(IntlkTrip.Disabled) OTE(Sts_IntlkTripDisabled) ,XIC(IntlkTrip.Inhibited) OTE(Sts_IntlkTripInhibited) ,XIC(IntlkTrip.Suppressed) OTE(Sts_IntlkTripSuppressed) ] ,[XIC(IntlkTrip.Ack) ,XIO(Cfg_HasIntlkTripAlm) ] OTE(Ack_IntlkTrip) ];
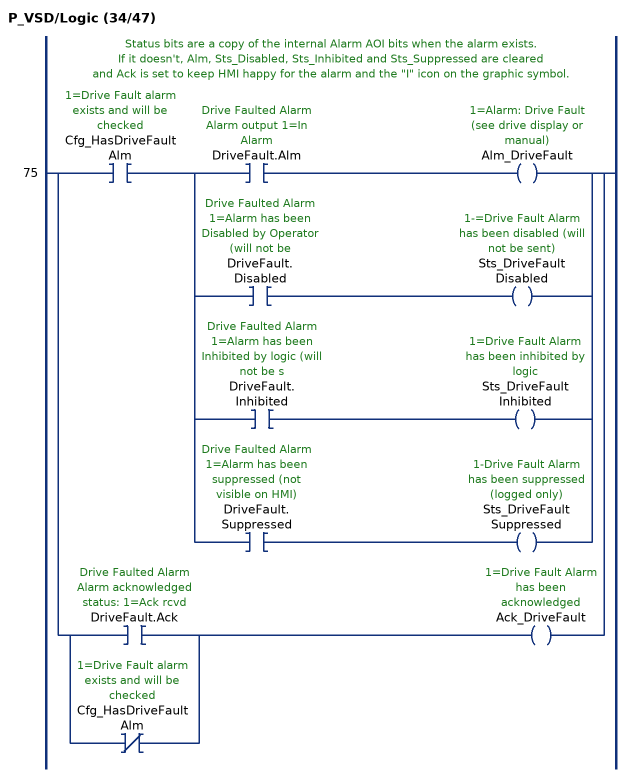
   // Status bits are a copy of the internal Alarm AOI bits when the alarm exists.
   // If it doesn't, Alm, Sts_Disabled, Sts_Inhibited and Sts_Suppressed are cleared
   // and Ack is set to keep HMI happy for the alarm and the "I" icon on the graphic symbol.
   75: [XIC(Cfg_HasDriveFaultAlm) [XIC(DriveFault.Alm) OTE(Alm_DriveFault) ,XIC(DriveFault.Disabled) OTE(Sts_DriveFaultDisabled) ,XIC(DriveFault.Inhibited) OTE(Sts_DriveFaultInhibited) ,XIC(DriveFault.Suppressed) OTE(Sts_DriveFaultSuppressed) ] ,[XIC(DriveFault.Ack) ,XIO(Cfg_HasDriveFaultAlm) ] OTE(Ack_DriveFault) ];
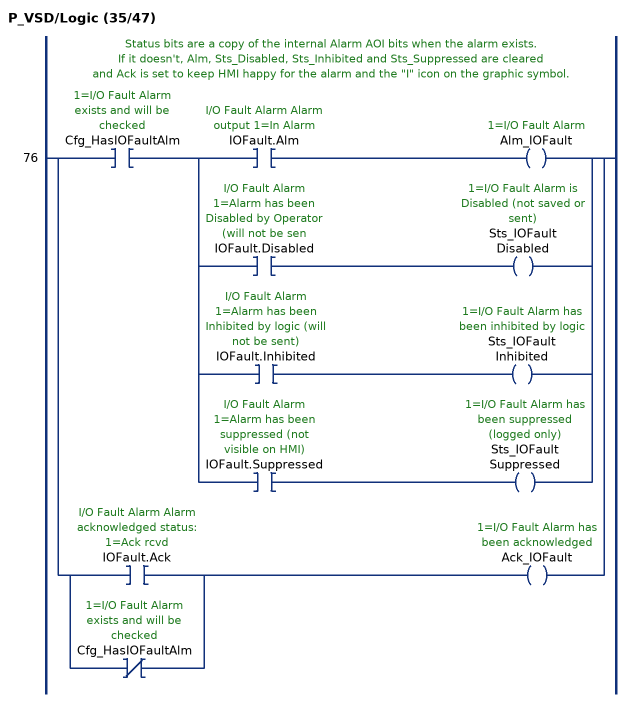
   // Status bits are a copy of the internal Alarm AOI bits when the alarm exists.
   // If it doesn't, Alm, Sts_Disabled, Sts_Inhibited and Sts_Suppressed are cleared
   // and Ack is set to keep HMI happy for the alarm and the "I" icon on the graphic symbol.
   76: [XIC(Cfg_HasIOFaultAlm) [XIC(IOFault.Alm) OTE(Alm_IOFault) ,XIC(IOFault.Disabled) OTE(Sts_IOFaultDisabled) ,XIC(IOFault.Inhibited) OTE(Sts_IOFaultInhibited) ,XIC(IOFault.Suppressed) OTE(Sts_IOFaultSuppressed) ] ,[XIC(IOFault.Ack) ,XIO(Cfg_HasIOFaultAlm) ] OTE(Ack_IOFault) ];
